TYPE DINT_INDEX : DINT(0..2147483647); END_TYPE

(* stored: Version 1.1.0.1
   DUT DINT_INDEX: Id {7106e443-8523-4f81-9862-83fecc04cc09} *)
